{attribute 'qualified_only'}
VAR_GLOBAL
  //-----------------------------------------------------------------------------
  // command and state structure
  //  - datafields for anyone to access
  //    - ADS via symbol
  //    - cyclic mapping to any other cyclic network/runtime
  //-----------------------------------------------------------------------------
  Ctrl                        : ARRAY[1..PLC_CONSTANT.MAX_AXIS] OF ST_FLY_CTRL;      // command structure to write into
  State                       : ARRAY[1..PLC_CONSTANT.MAX_AXIS] OF ST_FLY_STATE;     // state structure to read from


  //-----------------------------------------------------------------------------
  // data and info structure
  //  - parameter data fields for
  //    - Ctrl  --> Data
  //    - State --> Info
  //-----------------------------------------------------------------------------
//  Info                        : ARRAY[1..PLC_CONSTANT.MAX_AXIS] OF ST_FLY_INFO;
  Data                        : ARRAY[1..PLC_CONSTANT.MAX_AXIS] OF ST_FLY_DATA;


  //-----------------------------------------------------------------------------
  // R/W datafields
  // - optional data for CheckMask
  // - The Options contains two position values as limits. 
  //   The check for these position limits can be activated. 
  //   To do this, two flags 
  //   (GearInSync_CheckMask_OptionalMinPos, 
  //    GearInSync_CheckMask_OptionalMaxPos) 
  //   have to be set in the SyncMode structure.
  //
  //-----------------------------------------------------------------------------
  Options                     : ARRAY[1..PLC_CONSTANT.MAX_AXIS] OF ST_FLY_OPTIONS;

END_VAR

(* stored: Version 1.1.0.1
   GVL GVL_FLYING_SAW: Id {10ad4b33-a09a-4f46-807d-1c84a92fe04c} *)
